// TwinCAT 3 PLC project Test
// ProgramVersion: 3.1.4026.10
// libraries:
//   Tc2_Standard, * (Beckhoff Automation GmbH)
//   Tc2_System, * (Beckhoff Automation GmbH)
//   Tc3_Module, * (Beckhoff Automation GmbH)
// project tree:
//   GVLs/ GVL_Var.TcGVL
//   Util/ FlashBits.TcPOU, Pulser.TcPOU (not stored), TimeOut.TcPOU (not stored)
//   / PlcTask.TcTTO
//   POUs/ MAIN.TcPOU
//   SafetyLogic/ SafetyLogic.TcPOU
// real-time tasks:
//   TASK PlcTask: cycle T#10ms, priority 20, ADS port 350
// I/O:
//   DEVICE Device 1 (EtherCAT), AmsNetId 5.63.87.154.2.1
//     Term 7 (EK1200) [EK1200-5000 EtherCAT Power supply (2A E-Bus)]
//       Term 2 (EL1008) [EL1008 8Ch. Dig. Input 24V, 3ms]
//       Term 3 (EL2008) [EL2008 8Ch. Dig. Output 24V, 0.5A]
//       Term 4 (EL1918) [EL1918, 8Ch. Safety Input 24V, TwinSAFE]
//         modules: Module 2 (FSLOGIC)
//       Term 5 (EL2904) [EL2904, 4 Ch. Safety Output 24V, 0.5A, TwinSAFE]
//         modules: Module 1 (FSOES), Module 2 (DO)
//       Term 6 (EK1122) [EK1122 2 port EtherCAT junction]
//         Box 8 (FANUC R-30iB Plus) [FANUC R-30iB Plus]
//           modules: Module 1 (Robot FSoE)
// variable links:
//   Device 1 (EtherCAT) <-> Device 1 (EtherCAT)/Term 7 (EK1200)/Term 6 (EK1122)/Box 8 (FANUC R-30iB Plus)
//     Term 7 (EK1200)/Term 4 (EL1918)/ConnectionInputs/TwinSafeGroup1.0x000100C4 - Robot FSoE (Robot FSoE)_1_3 TxPDO <-> Module 1 (Robot FSoE)/Outputs/FSOE
//     Term 7 (EK1200)/Term 4 (EL1918)/ConnectionOutputs/TwinSafeGroup1.0x000100C4 - Robot FSoE (Robot FSoE)_1_3 RxPDO <-> Module 1 (Robot FSoE)/Inputs/FSOE
//   Test/Test Instance <-> Device 1 (EtherCAT)/Term 7 (EK1200)/Term 2 (EL1008)
//     PlcTask Inputs/SafetyLogic.iResetEstop <-> Channel 1/Input
//   Test/Test Instance <-> Device 1 (EtherCAT)/Term 7 (EK1200)/Term 3 (EL2008)
//     PlcTask Outputs/SafetyLogic.TurnOff <-> Channel 2/Output
//   Test/Test Instance <-> Device 1 (EtherCAT)/Term 7 (EK1200)/Term 4 (EL1918)
//     PlcTask Inputs/SafetyLogic.GroupComError <-> StandardInputs/TwinSafeGroup1.FromSafetyComError_8
//     PlcTask Outputs/SafetyLogic.ActivateEstop <-> StandardOutputs/TwinSafeGroup1.FromPlcActivateEstop_7
//     PlcTask Outputs/SafetyLogic.ErrorActknowledgement <-> StandardOutputs/TwinSafeGroup1.ErrorAcknowledgement_1
//     PlcTask Outputs/SafetyLogic.ResetSafety <-> StandardOutputs/TwinSafeGroup1.FromPlcResetEstop_5
//     PlcTask Outputs/SafetyLogic.SafetyRun <-> StandardOutputs/TwinSafeGroup1.Run_2
//   Test/Test Instance <-> Device 1 (EtherCAT)/Term 7 (EK1200)/Term 6 (EK1122)/Box 8 (FANUC R-30iB Plus)
//     PlcTask Inputs/GVL_Var.EthIB0 <-> IN128/DO[0]
//     PlcTask Outputs/GVL_Var.EthOB0 <-> OUT128/DI00[0]

CONFIGURATION Test
    RESOURCE PLC ON TwinCAT3
        TASK PlcTask(INTERVAL := T#10ms, PRIORITY := 20);
        PROGRAM MAIN WITH PlcTask : MAIN;
    END_RESOURCE
END_CONFIGURATION

// ---- GVLs/GVL_Var.TcGVL
{attribute 'qualified_only'}
VAR_GLOBAL
	EthIB0 AT %I* : UINT ;
	EthOB0 AT %Q* : UINT ;
END_VAR

// ---- POUs/MAIN.TcPOU
PROGRAM MAIN
VAR
	Input1 AT %I* : BOOL ;
	Output1 AT %Q* : BOOL ;
END_VAR

Output1 := Input1;

SafetyLogic();

Gvl_Var.EthOB0.1 := FlashBits.Bits.3;
Gvl_Var.EthOB0.2 := FlashBits.Bits.4;

END_PROGRAM

// ---- SafetyLogic/SafetyLogic.TcPOU
PROGRAM SafetyLogic
VAR
	SafetyRun AT %Q* : BOOL;
	ErrorActknowledgement AT %Q* : BOOL;
	ResetSafety AT %Q* : BOOL;
	TestOut1 AT %Q* : BOOL;
	TestIn1 AT %I* : BOOL;
	TurnOff AT %Q*  : BOOL;
	ResetEstop : BOOL;
	iResetEstop AT %I* : BOOL;
	ActivateEstop AT %Q* : BOOL;
	GroupComError AT %I* : BOOL;
END_VAR

SafetyRun := TRUE;
FlashBits();
IF (ResetEstop OR iResetEstop) THEN
	ErrorActknowledgement := FlashBits.Bits.3;
	ResetSafety:= FlashBits.Bits.3;
	Gvl_Var.EthOB0.0 := FlashBits.Bits.3;
ELSE
	ErrorActknowledgement := False;
	ResetSafety:= FALSE;
	Gvl_Var.EthOB0.0 := FALSE;	
END_IF

END_PROGRAM

// ---- Util/FlashBits.TcPOU
PROGRAM FlashBits
VAR_OUTPUT
	Bits : BYTE;
END_VAR
VAR
	MaxFlashFreq	: TIME := T#100MS;
    FlashTimer		: TON;    // timeout timer 
END_VAR

FlashTimer(IN:=NOT FlashTimer.Q,PT:=MaxFlashFreq);
IF FlashTimer.Q THEN
	IF Bits=0 THEN
		Bits :=1;
	ELSE	
		Bits:=Bits+1;
	END_IF
END_IF

END_PROGRAM
